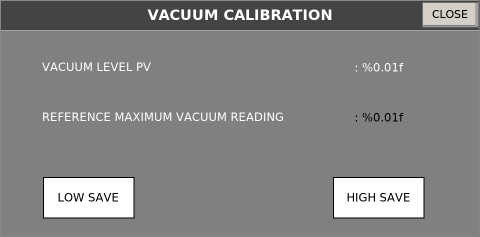
VISUALIZATION Vacuum_Calibration  // 480x237
    Rectangle (0,31 480x206)
    Rectangle (0,0 480x30), "VACUUM CALIBRATION"
    Label (39,47 129x40), "VACUUM LEVEL PV"
    Rectangle (336,44 86x47), ": %0.01f", text variable: ARrStnVacuumPV[6]
    Label (39,97 285x40), "REFERENCE MAXIMUM VACUUM READING"
    Rectangle (336,94 86x47), ": %0.01f", text variable: ARlrStnVacuumMaxReadSV[6]
        OnMouseDown: write the text variable via VisuDialogs.Numpad
    Rectangle (43,177 91x41), "LOW SAVE", colour toggle: ARbStnLowVacuumLvlSave[6]
        tap ARbStnLowVacuumLvlSave[6]
    Rectangle (333,177 91x41), "HIGH SAVE", colour toggle: ARbStnHighVacuumLvlSave[6]
        tap ARbStnHighVacuumLvlSave[6]
    Button (422,2 56x25), "CLOSE"
        toggle bManualCalibratePageOn
END_VISUALIZATION

(* stored: Version 1.1.0.1, ProductVersion 3.1.4024.12
   Visu Vacuum_Calibration: Id {c138b474-1ec5-4cc5-9651-3bc8c90dcab2} *)
